FUNCTION_BLOCK E_SEL_WSTRING (* Event-driven WSTRING selection *)
  (* Standard: 61499-1; Classification: Math; Function: Event-driven selection *)
  (* Version 0.1, 2001-11-27, JHC, Rockwell Automation, Moved to fb.rt.math. *)
  (* Version 0.0, 2001-04-12, JHC, Rockwell Automation, First XML version. *)
  (* Compiler header: package fb.rt.math; *)
  (* Compiler Java IBM VisualAge 3.0 *)
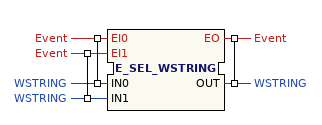
  EVENT_INPUT
    EI0 WITH IN0; (* Select INO *)
    EI1 WITH IN1; (* Select INO *)
  END_EVENT
  EVENT_OUTPUT
    EO WITH OUT; (* New selection event *)
  END_EVENT
  VAR_INPUT
    IN0 : WSTRING; (* Selected by EI0 *)
    IN1 : WSTRING; (* Selected by EI1 *)
  END_VAR
  VAR_OUTPUT
    OUT : WSTRING; (* Selected value *)
  END_VAR
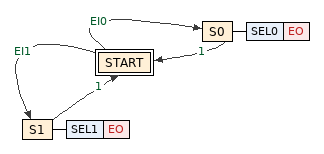
  EC_STATES
    START; (* Initial State *)
    S0 : SEL0 -> EO; (* Select IN0 *)
    S1 : SEL1 -> EO; (* Select IN1 *)
  END_STATES
  EC_TRANSITIONS
    START TO S0 := EI0;
    S0 TO START := 1;
    START TO S1 := EI1;
    S1 TO START := 1;
  END_TRANSITIONS
  ALGORITHM SEL0 IN ST:
OUT:=IN0;
  END_ALGORITHM
  ALGORITHM SEL1 IN ST:
OUT:=IN1;
  END_ALGORITHM
END_FUNCTION_BLOCK
